PROGRAM MAIN
VAR
	InputOutputConvert: InputOutputConvert;
	PID: PID;
	ElectricBox: ElectricBox;
END_VAR

ModbusRead();
ModbusWrite();
InputOutputConvert();
PID();
ElectricBox();

END_PROGRAM

(* stored: Version 1.1.0.1, ProductVersion 3.1.4024.6
   POU MAIN: Id {c4a70cbf-fcee-40e7-9278-ab5cba9e5400}, SpecialFunc None *)
